# EPICS substitutions: GALILMUL/GALILMUL-IOC-01App/Db/galil_profileMoveController.substitutions
file "$(MOTOR)/db/profileMoveController.template"
{
pattern
{P,       R,      PORT,   NAXES, NPOINTS, NPULSES,  TIMEOUT}
{"\$(P)DMC\$(CCP):", Prof1:, Galil,  8,     1441,    1441,     1}
}

file "$(GALIL)/GalilSup/Db/galil_profileMoveController.template"
{
pattern
{P,       R,      PORT,   TIMEOUT}
{"\$(P)DMC\$(CCP):",  Prof1:, Galil,  1}
}
